// TIA Portal V16 export
// export: Created 2021-04-06T19:52:16.3071342Z, ExportSetting WithDefaults, DisplayName Totally Integrated Automation Portal, DisplayVersion V16, DisplayName TIA Portal Version Control Interface, DisplayVersion V16, DisplayName TIA Portal Openness, DisplayVersion V16, DisplayName STEP 7 Professional, DisplayVersion V16, DisplayName STEP 7 Safety, DisplayVersion V16, DisplayName WinCC Unified SCADA Engineering System, DisplayVersion V16
DATA_BLOCK "modbus_FB_DB"   // DB3
VERSION : 0.1
// stored: AutoNumber true, DBAccessibleFromOPCUA true, InstanceOfName modbus_FB, InstanceOfType FB
"modbus_FB"
   // VAR_IN_OUT
   //    currentWeight : Array[0..12] of Real;
   // END_VAR
   // VAR
   //    MODBUS_ADDRESS : Array[0..12] of UInt;
   //    modbus_SenecaConnectPort1_FB { S7_SetPoint := 'True'} : "modbus_SenecaConnectPort1";
   //    modbus_SenecaConnectPort2_FB { S7_SetPoint := 'True'} : "modbus_SenecaConnectPort2";
   // END_VAR
BEGIN
END_DATA_BLOCK
